TYPE TC_config :
STRUCT
	iRawCountIn	AT %I*	: INT; 
	rTempC				: REAL;
	rTempF				: REAL;
END_STRUCT
END_TYPE

(* stored: Version 1.1.0.1, ProductVersion 3.1.4024.12
   DUT TC_config: Id {6fa5471c-063b-44ac-ad76-09eb605931bd} *)
